FUNCTION_BLOCK STankOut (* Basic Function Block Type *)
  (* Standard: 61499-2 *)
  (* Version 0.0, 2019-06-19, 4DIAC-IDE, 4DIAC-Consortium *)
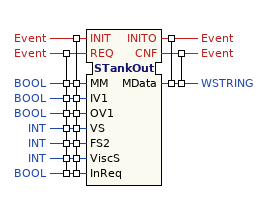
  EVENT_INPUT
    INIT WITH OV1, VS, FS2, MM, IV1, ViscS, InReq; (* Initialization Request *)
    REQ WITH OV1, VS, FS2, MM, IV1, ViscS, InReq; (* Normal Execution Request *)
  END_EVENT
  EVENT_OUTPUT
    INITO WITH MData; (* Initialization Confirm *)
    CNF WITH MData; (* Execution Confirmation *)
  END_EVENT
  VAR_INPUT
    MM : BOOL;
    IV1 : BOOL;
    OV1 : BOOL; (* Input event qualifier *)
    VS : INT;
    FS2 : INT;
    ViscS : INT;
    InReq : BOOL;
  END_VAR
  VAR_OUTPUT
    MData : WSTRING; (* Output event qualifier *)
  END_VAR
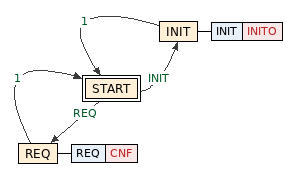
  EC_STATES
    START; (* Initial State *)
    INIT : INIT -> INITO; (* Initialization *)
    REQ : REQ -> CNF; (* Normal execution *)
  END_STATES
  EC_TRANSITIONS
    START TO INIT := INIT;
    INIT TO START := 1;
    START TO REQ := REQ;
    REQ TO START := 1;
  END_TRANSITIONS
  ALGORITHM INIT IN ST: (* Initialization algorithm *)

  END_ALGORITHM
  ALGORITHM REQ IN ST: (* Normally executed algorithm *)

  END_ALGORITHM
END_FUNCTION_BLOCK
